{attribute 'GeneratedUsingTerminal: EJ7334-0008-0016'}
{attribute addProperty BoxType "EJ7334-0008-0016"}
{attribute addProperty Id "StatusAT %I*Status_2569232E8"}
{attribute addProperty CRC "1163009244"}
{attribute addProperty Size "8"}
TYPE DCM_Status_Channel_45521CDC :
STRUCT
	{attribute addProperty Name "Status"}
	Status AT %I* : Status_2569232E;
END_STRUCT
END_TYPE

(* stored: Version 1.2.0.0, ProductVersion 3.1.4024.9
   DUT DCM_Status_Channel_45521CDC: Id {c386c5cf-c2d4-4924-af6a-c9f8794b7c81} *)
